KUKA KRL program: p01drop1_s1.src, p01drop1_s1.dat

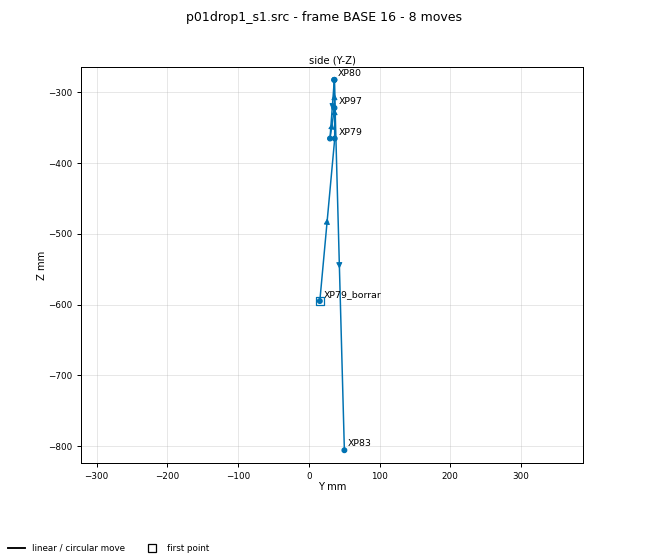
[picture p0: tool path of p01drop1_s1.src in frame BASE 16, 8 of 12 moves have a stored position in this frame; points joined in program order, loops and branches not executed]
--- p01drop1_s1.src ---
&ACCESS RVO1
&REL 4753
&PARAM EDITMASK = *
DEF p01drop1_s1( )

;================================================
; MODELO   : BALANCINA VIEJA
; IE GRUPO : FIP
; ESTACION : ST101
; ROBOT    : 101R1
; FUNCION  : DROP IP
;================================================

;FOLD INI
  ;FOLD BASISTECH INI
    GLOBAL INTERRUPT DECL 3 WHEN $STOPMESS==TRUE DO IR_STOPM ( )
    INTERRUPT ON 3
    BAS (#INITMOV,0 )
  ;ENDFOLD (BASISTECH INI)
;FOLD SPOTTECH INI
;USERSPOT(#INIT)
;ENDFOLD (SPOTTECH INI)
;FOLD GRIPPERTECH INI
USER_GRP(0,DUMMY,DUMMY,GDEFAULT)
INTERRUPT DECL 20 WHEN $FLAG[20]==FALSE DO GRPS(#MON_ERR,20)
;ENDFOLD (GRIPPERTECH INI)
  ;FOLD USER INI
    ;Make your modifications here

  ;ENDFOLD (USER INI)
;ENDFOLD (INI)

;ENTRAR_DEDOS()
;CERRAR_DEDOS()
;ENTRAR_RODILLO()
;ABRIR_CILINDRO_IP()
;CLAMPAR_GONDOLA()
o_type_req=FALSE

;INICIALIZACION GRIPER

;wait area

;FOLD PTP P77 Vel=100 % PDAT22 Tool[13] Base[0];%{PE}%R 5.6.13,%MKUKATPBASIS,%CMOVE,%VPTP,%P 1:PTP, 2:P77, 3:, 5:100, 7:PDAT22
$BWDSTART=FALSE
PDAT_ACT=PPDAT22
FDAT_ACT=FP77
BAS(#PTP_PARAMS,100)
PTP XP77
;ENDFOLD
;FOLD FORDTECH.Area_Req 2 Safety Position, 0 Return To Home, 0 ;%{PE}%MKUKATPUSER
;Area_Req (2,0,0)
wait for $in[18]
$out[18]=false
;ENDFOLD

;TRAYECTORIA DE ENTRADA


;===========================================================
;POSICION FOTO 1 (selccionar esta linea para repetir foto 1)
;===========================================================
;FOLD OUT 38 'PETICION A DISPOSITIVO 6' State=FALSE ;%{PE}%R 5.6.13,%MKUKATPBASIS,%COUT,%VOUTX,%P 2:38, 3:PETICION A DISPOSITIVO 6, 5:FALSE, 6:
$OUT[38]=FALSE
;ENDFOLD
;wait for false


;FOLD PTP P85 Vel=100 % PDAT27 Tool[14]:camara Base[14]:ems_sup;%{PE}%R 5.6.13,%MKUKATPBASIS,%CMOVE,%VPTP,%P 1:PTP, 2:P85, 3:, 5:100, 7:PDAT27
$BWDSTART=FALSE
PDAT_ACT=PPDAT27
FDAT_ACT=FP85
BAS(#PTP_PARAMS,100)
PTP XP85
;ENDFOLD

;FOLD WAIT Time=0.3 sec;%{PE}%R 5.6.13,%MKUKATPBASIS,%CWAIT,%VWAIT,%P 2:0.3
WAIT SEC 0.3
;ENDFOLD

;CHEQUEO SEÑALES RESETEADAS
MAFELEC_TECH (#CHECK_RESET, 8,0,0)

;PIDE FOTO
;FOLD FORDTECH.Tool_Rel 2 ;%{PE}%MKUKATPUSER
TOOL_REL (2)
;ENDFOLD

;PIDE CORRECCIONES
MAFELEC_TECH (#TYPE, 8,0,0)

;EVALUA CORRECCIONES
SWITCH I_TYPE_INFO
CASE 2
o_type_req=FALSE
;FOLD FORDTECH.Tool_Req 2 ;%{PE}%MKUKATPUSER
TOOL_REQ (2)
;ENDFOLD
RECAZOEMS()
goto home
case 3
o_type_req=FALSE
rechazo_bal()
GOTO HOME
ENDSWITCH

;APLICA CORRECIONES A LA BASE
base_data[16]=base_data[14]
MAFELEC_TECH (#GET_CORR, 16,0,0)

tool_data[16]=tool_data[14]
;APLICA CORRECCION ANGULO A TOOL
MAFELEC_TECH (#GET_CORR_TOOL,16 ,0,0)

;REGISTRA CORRECCIONES
MAFELEC_TECH (#REG1, 8,0,0)

;FINALIZA PROCESO CORRECCIONES
o_type_req=false
wait for i_type_info==0
;FOLD FORDTECH.Tool_Req 2 ;%{PE}%MKUKATPUSER
TOOL_REQ (2)
;ENDFOLD

;PUNTO SEGUNA FOTO
xP76=xP85
;FOLD PTP P76 Vel=100 % PDAT21 Tool[16]:camara_corregida Base[16]:EMS_SUP_CORREGIDA;%{PE}%R 5.6.13,%MKUKATPBASIS,%CMOVE,%VPTP,%P 1:PTP, 2:P76, 3:, 5:100, 7:PDAT21
$BWDSTART=FALSE
PDAT_ACT=PPDAT21
FDAT_ACT=FP76
BAS(#PTP_PARAMS,100)
PTP XP76
;ENDFOLD

;FOLD WAIT Time=0.3 sec;%{PE}%R 5.6.13,%MKUKATPBASIS,%CWAIT,%VWAIT,%P 2:0.3
WAIT SEC 0.3
;ENDFOLD

;PETICION SEGUNDA FOTO
;FOLD FORDTECH.Tool_Rel 6 ;%{PE}%MKUKATPUSER
TOOL_REL (6)
;ENDFOLD

;PETICION RESULTADO FOTO
MAFELEC_TECH (#TYPE, 8,0,0)

;EVALUA RESULTADO
SWITCH I_TYPE_INFO
CASE 1 ;FOTO OK
o_type_req=false
wait for i_type_info==0
CASE 2
o_type_req=FALSE
;FOLD FORDTECH.Tool_Req 6 ;%{PE}%MKUKATPUSER
TOOL_REQ (6)
;ENDFOLD
;wait for false
RECAZOEMS()
GOTO HOME
case 3
o_type_req=FALSE
rechazo_bal()
goto home
ENDSWITCH

;FINALIZA PROCESO SEGUNDA FOTO
;FOLD FORDTECH.Tool_Req 6 ;%{PE}%MKUKATPUSER
TOOL_REQ (6)
;ENDFOLD

if not i_dry then

;FOLD CHEQUEO LIMITE SEGUNDO OFFSET
;WAIT FOR EMSupbase_OFFSETz>-200
;WAIT FOR EMSupbase_OFFSETz<200
;WAIT FOR EMSupbase_OFFSETx>-200
;WAIT FOR EMSupbase_OFFSETx<200
;WAIT FOR EMSupbase_OFFSETb>-0.400
;WAIT FOR EMSupbase_OFFSETb<0.400
;ENDFOLD
;APLICAMOS OFFSET
;FOLD OFFSET CORR
;BASE_DATA[8].Z=EMSupbase_CORR.Z+EMSupbase_OFFSETz
;BASE_DATA[8].X=EMSupbase_CORR.X+EMSupbase_OFFSETx
;BASE_DATA[8].B=EMSupbase_CORR.B+EMSupbase_OFFSETb
;ENDFOLD
;goto alejandro
;SACAR_DEDOS()
;wait for false

;ACTIVAR TORQ MONITORING
;FOLD TORQMON SetLimits Axis 1: 50 % Axis 2: 40 % Axis 3: 40 % Axis 4: 50 % Axis 5: 40 % Axis 6: 40 %;%{PE}%R 5.6.13,%MKUKATPBASIS,%CTQ_MON,%VTQ_LIMITS,%P 2:TQ_LIMITS, 4:50, 7:40, 10:40, 13:50, 16:40, 19:40
SET_TQ_VALUES (50,40,40,50,40,40)
;ENDFOLD

;TRAYECTORIA ENTRADA A COGIDA

;FOLD LIN P79_borrar Vel=2 m/s CPDAT21 Tool[16]:camara_corregida Base[16]:EMS_SUP_CORREGIDA;%{PE}%R 5.6.13,%MKUKATPBASIS,%CMOVE,%VLIN,%P 1:LIN, 2:P79_borrar, 3:, 5:2, 7:CPDAT21
$BWDSTART=FALSE
LDAT_ACT=LCPDAT21
FDAT_ACT=FP79_borrar
BAS(#CP_PARAMS,2)
LIN XP79_borrar
;ENDFOLD

;FOLD LIN P79 Vel=2 m/s CPDAT10 Tool[16]:camara_corregida Base[16]:EMS_SUP_CORREGIDA;%{PE}%R 5.6.13,%MKUKATPBASIS,%CMOVE,%VLIN,%P 1:LIN, 2:P79, 3:, 5:2, 7:CPDAT10
$BWDSTART=FALSE
LDAT_ACT=LCPDAT10
FDAT_ACT=FP79
BAS(#CP_PARAMS,2)
LIN XP79
;ENDFOLD

;ABRE CLAMPAS
ABRIR_DEDOS()

;MOVIMIENTO A PUNTO DEJADA
if false then
;FOLD LIN P80 Vel=2 m/s CPDAT11 Tool[16]:camara_corregida Base[16]:EMS_SUP_CORREGIDA;%{PE}%R 5.6.13,%MKUKATPBASIS,%CMOVE,%VLIN,%P 1:LIN, 2:P80, 3:, 5:2, 7:CPDAT11
$BWDSTART=FALSE
LDAT_ACT=LCPDAT11
FDAT_ACT=FP80
BAS(#CP_PARAMS,2)
LIN XP80
;ENDFOLD
endif

;FOLD LIN P98 Vel=2 m/s CPDAT18 Tool[16]:camara_corregida Base[16]:EMS_SUP_CORREGIDA;%{PE}%R 5.6.13,%MKUKATPBASIS,%CMOVE,%VLIN,%P 1:LIN, 2:P98, 3:, 5:2, 7:CPDAT18
$BWDSTART=FALSE
LDAT_ACT=LCPDAT18
FDAT_ACT=FP98
BAS(#CP_PARAMS,2)
LIN XP98
;ENDFOLD
;FOLD LIN P97 Vel=2 m/s CPDAT17 Tool[16]:camara_corregida Base[16]:EMS_SUP_CORREGIDA;%{PE}%R 5.6.13,%MKUKATPBASIS,%CMOVE,%VLIN,%P 1:LIN, 2:P97, 3:, 5:2, 7:CPDAT17
$BWDSTART=FALSE
LDAT_ACT=LCPDAT17
FDAT_ACT=FP97
BAS(#CP_PARAMS,2)
LIN XP97
;ENDFOLD

;FOLD LIN P95 Vel=1 m/s CPDAT15 Tool[16]:camara_corregida Base[16]:EMS_SUP_CORREGIDA;%{PE}%R 5.6.13,%MKUKATPBASIS,%CMOVE,%VLIN,%P 1:LIN, 2:P95, 3:, 5:1, 7:CPDAT15
$BWDSTART=FALSE
LDAT_ACT=LCPDAT15
FDAT_ACT=FP95
BAS(#CP_PARAMS,1)
LIN XP95
;ENDFOLD

;CIERRA CLAMPAS
if not B_EMSdry then
CERRAR_DEDOS()
endif

;FOLD WAIT Time=1 sec;%{PE}%R 5.6.13,%MKUKATPBASIS,%CWAIT,%VWAIT,%P 2:1
WAIT SEC 1
;ENDFOLD

;FOLD LIN P96 Vel=1 m/s CPDAT16 Tool[16]:camara_corregida Base[16]:EMS_SUP_CORREGIDA;%{PE}%R 5.6.13,%MKUKATPBASIS,%CMOVE,%VLIN,%P 1:LIN, 2:P96, 3:, 5:1, 7:CPDAT16
$BWDSTART=FALSE
LDAT_ACT=LCPDAT16
FDAT_ACT=FP96
BAS(#CP_PARAMS,1)
LIN XP96
;ENDFOLD

IF false THEN
;CHEQUEA CLAMPAS CERRADAS
ENDIF
if false then
endif

;ESPERA RESULTADOS CAMARAS ACIMUT Y VOLANTE
;FOLD FORDTECH.Tool_Rel 3 ;%{PE}%MKUKATPUSER
TOOL_REL (3)
;ENDFOLD
;FOLD FORDTECH.Tool_Req 3 ;%{PE}%MKUKATPUSER
TOOL_REQ (3)
;ENDFOLD

if not B_EMSdry then
;ABRE GARRA PARA SOLTAR IP

ABRIR_CILINDRO_IP()
endif

if B_EMSdry then
;punto interdio para liberar orejetas
endif

;FOLD LIN P83 Vel=1 m/s CPDAT13 Tool[16]:camara_corregida Base[16]:EMS_SUP_CORREGIDA;%{PE}%R 5.6.13,%MKUKATPBASIS,%CMOVE,%VLIN,%P 1:LIN, 2:P83, 3:, 5:1, 7:CPDAT13
$BWDSTART=FALSE
LDAT_ACT=LCPDAT13
FDAT_ACT=FP83
BAS(#CP_PARAMS,1)
LIN XP83
;ENDFOLD
;MOVIMIENTO SALIDA
alejandro:

endif

if i_dry then
;FOLD FORDTECH.Tool_Rel 3 ;%{PE}%MKUKATPUSER
TOOL_REL (3)
;ENDFOLD
;FOLD FORDTECH.Tool_Req 3 ;%{PE}%MKUKATPUSER
TOOL_REQ (3)
;ENDFOLD
endif

;DEJA TORQ MONITORING EN VALORES NOMINALES
;FOLD TORQMON SetDefault;%{PE}%R 5.6.13,%MKUKATPBASIS,%CTQ_MON,%VTQ_DEFAULT,%P 2:TQ_DEFAULT
SET_TQ_VALUES ( )
;ENDFOLD

;TRAYECTORIA SALIDA AREA

;wait area ems
;FOLD PTP P89 Vel=100 % PDAT30 Tool[12] Base[0];%{PE}%R 5.6.13,%MKUKATPBASIS,%CMOVE,%VPTP,%P 1:PTP, 2:P89, 3:, 5:100, 7:PDAT30
$BWDSTART=FALSE
PDAT_ACT=PPDAT30
FDAT_ACT=FP89
BAS(#PTP_PARAMS,100)
PTP XP89
;ENDFOLD

;AREA LIBRE Y TRABAJO REALIZADO
;FOLD FORDTECH.Job_Rdy 2 , 1 ;%{PE}%MKUKATPUSER
JOB_READY (2,1)
;ENDFOLD
;FOLD FORDTECH.Area_Rel 2 ;%{PE}%MKUKATPUSER
AREA_REL (2)
;ENDFOLD




home:


END

--- p01drop1_s1.dat ---
&ACCESS RVO1
&REL 4753
&PARAM EDITMASK = *
DEFDAT  P01DROP1_S1
;FOLD EXTERNAL DECLARATIONS;%{PE}%MKUKATPBASIS,%CEXT,%VCOMMON,%P
;FOLD GRIPPERTECH EXT
EXT  H50 (INT  :IN,INT  :IN,INT  :IN,GRP_TYP  :IN )
;ENDFOLD (GRIPPERTECH EXT)
;FOLD SPOTTECH EXT
EXT  USERSPOT (S_COMMAND  :IN,SPOT_TYPE  :IN )
;ENDFOLD (SPOTTECH EXT)
;FOLD BASISTECH EXT;%{PE}%MKUKATPBASIS,%CEXT,%VEXT,%P
EXT  BAS (BAS_COMMAND  :IN,REAL  :IN )
DECL INT SUCCESS
;ENDFOLD (BASISTECH EXT)
;FOLD USER EXT;%{E}%MKUKATPUSER,%CEXT,%VEXT,%P
;Make here your modifications

;ENDFOLD (USER EXT)
;ENDFOLD (EXTERNAL DECLARATIONS)
DECL BASIS_SUGG_T LAST_BASIS={POINT1[] "P100b                   ",POINT2[] "P100b                   ",CP_PARAMS[] "CPDAT21                 ",PTP_PARAMS[] "PDAT36                  ",CONT[] "                        ",CP_VEL[] "2                       ",PTP_VEL[] "100                     ",SYNC_PARAMS[] "SYNCDAT                 ",SPL_NAME[] "S0                      "}
DECL E6POS XP1={X 1562.28699,Y 893.286072,Z 1286.09595,A -15.2613897,B 0.657847583,C -90.4761429,S 2,T 3,E1 0.0,E2 0.0,E3 0.0,E4 0.0,E5 0.0,E6 0.0}
DECL FDAT FP1={TOOL_NO 10,BASE_NO 0,IPO_FRAME #BASE,POINT2[] " ",TQ_STATE FALSE}
DECL PDAT PPDAT1={VEL 100.0,ACC 100.0,APO_DIST 100.0,APO_MODE #CPTP}
DECL E6POS XP2={X 0.052320879,Y -135.084106,Z 32.6104889,A 0.252467006,B -0.648865819,C 1.13480794,S 2,T 3,E1 0.0,E2 0.0,E3 0.0,E4 0.0,E5 0.0,E6 0.0}
DECL FDAT FP2={TOOL_NO 10,BASE_NO 8,IPO_FRAME #BASE,POINT2[] " ",TQ_STATE FALSE}
DECL PDAT PPDAT2={VEL 100.0,ACC 100.0,APO_DIST 100.0}
DECL E6POS XP3={X -0.226943403,Y -135.580994,Z 57.4539795,A 0.252323091,B -0.648702681,C 1.13486397,S 2,T 3,E1 0.0,E2 0.0,E3 0.0,E4 0.0,E5 0.0,E6 0.0}
DECL FDAT FP3={TOOL_NO 10,BASE_NO 8,IPO_FRAME #BASE,POINT2[] " ",TQ_STATE FALSE}
DECL PDAT PPDAT3={VEL 100.0,ACC 100.0,APO_DIST 100.0}
DECL E6POS XP4={X 917.980408,Y 1082.76501,Z 1563.30298,A -10.58006,B -0.816496015,C -90.0786209,S 2,T 3,E1 0.0,E2 0.0,E3 0.0,E4 0.0,E5 0.0,E6 0.0}
DECL FDAT FP4={TOOL_NO 3,BASE_NO 0,IPO_FRAME #BASE,POINT2[] " ",TQ_STATE FALSE}
DECL PDAT PPDAT4={VEL 100.0,ACC 100.0,APO_DIST 100.0,APO_MODE #CPTP}
DECL PDAT PPDAT5={VEL 100.0,ACC 100.0,APO_DIST 100.0}
DECL E6POS XP55={X 669.274719,Y 1258.45898,Z 1571.16199,A 1.68324995,B 0.417000502,C -88.9230118,S 2,T 11,E1 0.0,E2 0.0,E3 0.0,E4 0.0,E5 0.0,E6 0.0}
DECL FDAT FP55={TOOL_NO 3,BASE_NO 0,IPO_FRAME #BASE,POINT2[] " ",TQ_STATE FALSE}
DECL PDAT PPDAT6={VEL 100.0,ACC 100.0,APO_DIST 100.0}
DECL LDAT LCPDAT3={VEL 2.0,ACC 100.0,APO_DIST 100.0,APO_FAC 50.0,ORI_TYP #VAR,CIRC_TYP #BASE,JERK_FAC 50.0,EXAX_IGN 0}
DECL E6POS XP56={X 3.78204703,Y -128.492996,Z -299.213898,A 0.252413303,B -0.64881891,C 1.13486505,S 2,T 3,E1 0.0,E2 0.0,E3 0.0,E4 0.0,E5 0.0,E6 0.0}
DECL FDAT FP56={TOOL_NO 10,BASE_NO 8,IPO_FRAME #BASE,POINT2[] " ",TQ_STATE FALSE}
DECL PDAT PPDAT7={VEL 100.0,ACC 100.0,APO_DIST 50.0,APO_MODE #CPTP}
DECL E6POS XP57={X 825.400024,Y 974.496826,Z 1563.53699,A -6.83336401,B -0.817213476,C -90.0786514,S 2,T 3,E1 0.0,E2 0.0,E3 0.0,E4 0.0,E5 0.0,E6 0.0}
DECL FDAT FP57={TOOL_NO 3,BASE_NO 0,IPO_FRAME #BASE,POINT2[] " ",TQ_STATE FALSE}
DECL PDAT PPDAT8={VEL 100.0,ACC 100.0,APO_DIST 100.0}
DECL LDAT LCPDAT1={VEL 2.0,ACC 100.0,APO_DIST 100.0,APO_FAC 50.0,ORI_TYP #VAR,CIRC_TYP #BASE,JERK_FAC 50.0,EXAX_IGN 0}
DECL E6POS XP58={X 6.92813683,Y -122.939102,Z -579.260681,A 0.251890212,B -0.648669422,C 1.13512194,S 2,T 11,E1 0.0,E2 0.0,E3 0.0,E4 0.0,E5 0.0,E6 0.0}
DECL FDAT FP58={TOOL_NO 3,BASE_NO 8,IPO_FRAME #BASE,POINT2[] " ",TQ_STATE FALSE}
DECL LDAT LCPDAT2={VEL 2.0,ACC 100.0,APO_DIST 100.0,APO_FAC 50.0,ORI_TYP #VAR,CIRC_TYP #BASE,JERK_FAC 50.0,EXAX_IGN 0}
DECL E6POS XP59={X 1195.93005,Y 946.286804,Z 1558.15601,A -25.4987297,B -0.698007703,C -90.0127335,S 2,T 3,E1 0.0,E2 0.0,E3 0.0,E4 0.0,E5 0.0,E6 0.0}
DECL FDAT FP59={TOOL_NO 3,BASE_NO 0,IPO_FRAME #BASE,POINT2[] " ",TQ_STATE FALSE}
DECL PDAT PPDAT9={VEL 100.0,ACC 100.0,APO_DIST 100.0,APO_MODE #CPTP}
DECL E6POS XP60={X 1607.74902,Y 781.598511,Z 1575.47095,A -48.1744194,B -1.694278,C -88.870842,S 2,T 2,E1 0.0,E2 0.0,E3 0.0,E4 0.0,E5 0.0,E6 0.0}
DECL FDAT FP60={TOOL_NO 3,BASE_NO 0,IPO_FRAME #BASE,POINT2[] " ",TQ_STATE FALSE}
DECL PDAT PPDAT10={VEL 100.0,ACC 100.0,APO_DIST 100.0,APO_MODE #CPTP}
DECL E6POS XP61={X 2.21973109,Y 78.0449219,Z -473.749786,A 0.453805208,B -1.02935696,C 1.12841296,S 2,T 11,E1 0.0,E2 0.0,E3 0.0,E4 0.0,E5 0.0,E6 0.0}
DECL FDAT FP61={TOOL_NO 10,BASE_NO 6,IPO_FRAME #BASE,POINT2[] " ",TQ_STATE FALSE}
DECL PDAT PPDAT11={VEL 100.0,ACC 100.0,APO_DIST 100.0}
DECL E6POS XP62={X 686.276306,Y 1072.54199,Z 1338.49402,A -3.73349309,B -0.516365111,C -90.2921371,S 2,T 3,E1 0.0,E2 0.0,E3 0.0,E4 0.0,E5 0.0,E6 0.0}
DECL FDAT FP62={TOOL_NO 10,BASE_NO 0,IPO_FRAME #BASE,POINT2[] " ",TQ_STATE FALSE}
DECL PDAT PPDAT12={VEL 100.0,ACC 100.0,APO_DIST 100.0,APO_MODE #CPTP}
DECL E6POS XP63={X 4.17468405,Y -128.584198,Z -273.346893,A 0.318527609,B -0.649609089,C 1.13304698,S 2,T 11,E1 0.0,E2 0.0,E3 0.0,E4 0.0,E5 0.0,E6 0.0}
DECL FDAT FP63={TOOL_NO 3,BASE_NO 8,IPO_FRAME #BASE,POINT2[] " ",TQ_STATE FALSE}
DECL PDAT PPDAT13={VEL 100.0,ACC 100.0,APO_DIST 100.0,APO_MODE #CPTP}
DECL E6POS XP64={X 141.040298,Y -131.536896,Z -626.476685,A -0.01522478,B 7.10692596,C 0.110732399,S 2,T 3,E1 0.0,E2 0.0,E3 0.0,E4 0.0,E5 0.0,E6 0.0}
DECL FDAT FP64={TOOL_NO 3,BASE_NO 8,IPO_FRAME #BASE,POINT2[] " ",TQ_STATE FALSE}
DECL PDAT PPDAT14={VEL 100.0,ACC 100.0,APO_DIST 100.0,APO_MODE #CPTP}
DECL E6POS XP65={X 1145.12195,Y 865.575378,Z 1562.22705,A -24.1379299,B -0.725280404,C -90.2146072,S 2,T 2,E1 0.0,E2 0.0,E3 0.0,E4 0.0,E5 0.0,E6 0.0}
DECL FDAT FP65={TOOL_NO 3,BASE_NO 0,IPO_FRAME #BASE,POINT2[] " ",TQ_STATE FALSE}
DECL PDAT PPDAT15={VEL 100.0,ACC 100.0,APO_DIST 100.0,APO_MODE #CPTP}
DECL E6POS XP66={X 2.245502,Y 78.0254288,Z -473.714996,A 0.452297091,B -1.028229,C 1.12880397,S 2,T 11,E1 0.0,E2 0.0,E3 0.0,E4 0.0,E5 0.0,E6 0.0}
DECL FDAT FP66={TOOL_NO 10,BASE_NO 8,IPO_FRAME #BASE,POINT2[] " ",TQ_STATE FALSE}
DECL PDAT PPDAT16={VEL 100.0,ACC 100.0,APO_DIST 100.0,APO_MODE #CPTP}
DECL E6POS XP67={X 0.474618286,Y -135.130203,Z 56.3668594,A 0.318735003,B -0.650003672,C 1.133497,S 2,T 3,E1 0.0,E2 0.0,E3 0.0,E4 0.0,E5 0.0,E6 0.0}
DECL FDAT FP67={TOOL_NO 3,BASE_NO 8,IPO_FRAME #BASE,POINT2[] " ",TQ_STATE FALSE}
DECL LDAT LCPDAT4={VEL 2.0,ACC 100.0,APO_DIST 100.0,APO_FAC 50.0,ORI_TYP #VAR,CIRC_TYP #BASE,JERK_FAC 50.0,EXAX_IGN 0}
DECL E6POS XP68={X 2.50332093,Y -131.528702,Z -125.126297,A 0.318527102,B -0.649853289,C 1.13311696,S 2,T 11,E1 0.0,E2 0.0,E3 0.0,E4 0.0,E5 0.0,E6 0.0}
DECL FDAT FP68={TOOL_NO 3,BASE_NO 8,IPO_FRAME #BASE,POINT2[] " ",TQ_STATE FALSE}
DECL LDAT LCPDAT5={VEL 2.0,ACC 100.0,APO_DIST 100.0,APO_FAC 50.0,ORI_TYP #VAR,CIRC_TYP #BASE,JERK_FAC 50.0,EXAX_IGN 0}
DECL E6POS XP69={X 2768.47705,Y 6.94654799,Z 2006.30298,A -150.0289,B 15.6658697,C -84.9255676,S 2,T 43,E1 0.0,E2 0.0,E3 0.0,E4 0.0,E5 0.0,E6 0.0}
DECL FDAT FP69={TOOL_NO 3,BASE_NO 0,IPO_FRAME #BASE,POINT2[] " ",TQ_STATE FALSE}
DECL PDAT PPDAT17={VEL 100.0,ACC 100.0,APO_DIST 100.0,APO_MODE #CPTP}
DECL E6POS XP70={X 2181.64502,Y 940.81012,Z 1193.08899,A -55.6323204,B 0.397260487,C -90.4529495,S 2,T 10,E1 0.0,E2 0.0,E3 0.0,E4 0.0,E5 0.0,E6 0.0}
DECL FDAT FP70={TOOL_NO 10,BASE_NO 0,IPO_FRAME #BASE,POINT2[] " ",TQ_STATE FALSE}
DECL PDAT PPDAT18={VEL 100.0,ACC 100.0,APO_DIST 100.0,APO_MODE #CPTP}
DECL E6POS XP71={X 682.504395,Y 1586.74194,Z 1564.78699,A 0.650965273,B -0.740677118,C -89.7750626,S 2,T 3,E1 0.0,E2 0.0,E3 0.0,E4 0.0,E5 0.0,E6 0.0}
DECL FDAT FP71={TOOL_NO 3,BASE_NO 0,IPO_FRAME #BASE,POINT2[] " ",TQ_STATE FALSE}
DECL LDAT LCPDAT7={VEL 2.0,ACC 100.0,APO_DIST 100.0,APO_FAC 50.0,ORI_TYP #VAR,CIRC_TYP #BASE,JERK_FAC 50.0,EXAX_IGN 0}
DECL LDAT LCPDAT8={VEL 2.0,ACC 100.0,APO_DIST 100.0,APO_FAC 50.0,ORI_TYP #VAR,CIRC_TYP #BASE,JERK_FAC 50.0,EXAX_IGN 0}
DECL E6POS XP72={X 0.052320879,Y -135.084106,Z 32.6104889,A 0.252467006,B -0.648865819,C 1.13480794,S 2,T 3,E1 0.0,E2 0.0,E3 0.0,E4 0.0,E5 0.0,E6 0.0}
DECL FDAT FP72={TOOL_NO 10,BASE_NO 8,IPO_FRAME #BASE,POINT2[] " ",TQ_STATE FALSE}
DECL E6POS XP73={X 0.149559602,Y -134.919601,Z 24.4487591,A 0.252554208,B -0.648425877,C 1.13475394,S 2,T 3,E1 0.0,E2 0.0,E3 0.0,E4 0.0,E5 0.0,E6 0.0}
DECL FDAT FP73={TOOL_NO 10,BASE_NO 8,IPO_FRAME #BASE,POINT2[] " ",TQ_STATE FALSE}
DECL LDAT LCPDAT9={VEL 2.0,ACC 100.0,APO_DIST 100.0,APO_FAC 50.0,ORI_TYP #VAR,CIRC_TYP #BASE,JERK_FAC 50.0,EXAX_IGN 0}
DECL E6POS XP74={X 177.492004,Y 2082.823,Z 1702.56897,A -0.50292927,B 45.5188103,C 179.499405,S 2,T 11,E1 0.0,E2 0.0,E3 0.0,E4 0.0,E5 0.0,E6 0.0}
DECL FDAT FP74={TOOL_NO 0,BASE_NO 0,IPO_FRAME #BASE,POINT2[] " ",TQ_STATE FALSE}
DECL PDAT PPDAT19={VEL 100.0,ACC 100.0,APO_DIST 100.0}
DECL E6POS XP75={X -125.971199,Y -265.283813,Z -316.319305,A 90.6103363,B -1.78813803,C -0.124596797,S 2,T 10,E1 0.0,E2 0.0,E3 0.0,E4 0.0,E5 0.0,E6 0.0}
DECL FDAT FP75={TOOL_NO 8,BASE_NO 14,IPO_FRAME #BASE,POINT2[] " ",TQ_STATE FALSE}
DECL PDAT PPDAT20={VEL 100.0,ACC 100.0,APO_DIST 100.0}
DECL E6POS XP76={X -128.091095,Y 0.680960417,Z -757.682922,A 89.7646408,B -0.642541885,C 0.220073298,S 2,T 11,E1 0.0,E2 0.0,E3 0.0,E4 0.0,E5 0.0,E6 0.0}
DECL FDAT FP76={TOOL_NO 16,BASE_NO 16,IPO_FRAME #BASE,POINT2[] " ",TQ_STATE FALSE}
DECL PDAT PPDAT21={VEL 100.0,ACC 100.0,APO_DIST 100.0}
DECL E6POS XP77={X 705.314392,Y 2000.59497,Z 1624.87805,A -13.2357502,B 44.7311783,C 178.321304,S 2,T 11,E1 0.0,E2 0.0,E3 0.0,E4 0.0,E5 0.0,E6 0.0}
DECL FDAT FP77={TOOL_NO 13,BASE_NO 0,IPO_FRAME #BASE,POINT2[] " ",TQ_STATE FALSE}
DECL PDAT PPDAT22={VEL 100.0,ACC 100.0,APO_DIST 100.0}
DECL E6POS XP78={X 224.640701,Y 2078.11694,Z 1675.72803,A -0.294790298,B 45.0043297,C 179.436996,S 2,T 11,E1 0.0,E2 0.0,E3 0.0,E4 0.0,E5 0.0,E6 0.0}
DECL FDAT FP78={TOOL_NO 0,BASE_NO 0,IPO_FRAME #BASE,POINT2[] " ",TQ_STATE FALSE}
DECL PDAT PPDAT23={VEL 100.0,ACC 100.0,APO_DIST 100.0}
DECL E6POS XP79={X -130.524094,Y 36.7159882,Z -365.105804,A 89.8188171,B -1.25319099,C 0.0377966203,S 2,T 11,E1 0.0,E2 0.0,E3 0.0,E4 0.0,E5 0.0,E6 0.0}
DECL FDAT FP79={TOOL_NO 16,BASE_NO 16,IPO_FRAME #BASE,POINT2[] " ",TQ_STATE FALSE}
DECL LDAT LCPDAT10={VEL 2.0,ACC 20.0,APO_DIST 100.0,APO_FAC 50.0,ORI_TYP #VAR,CIRC_TYP #BASE,JERK_FAC 50.0,EXAX_IGN 0}
DECL E6POS XP80={X -134.476898,Y 36.1417999,Z -282.15741,A 89.8160934,B -1.10210598,C -0.134312794,S 2,T 11,E1 0.0,E2 0.0,E3 0.0,E4 0.0,E5 0.0,E6 0.0}
DECL FDAT FP80={TOOL_NO 16,BASE_NO 16,IPO_FRAME #BASE,POINT2[] " ",TQ_STATE FALSE}
DECL LDAT LCPDAT11={VEL 2.0,ACC 20.0,APO_DIST 100.0,APO_FAC 50.0,ORI_TYP #VAR,CIRC_TYP #BASE,JERK_FAC 50.0,EXAX_IGN 0}
DECL E6POS XP81={X 2576.92993,Y -773.447327,Z -3076.573,A 88.4551315,B -0.226906598,C 91.8414612,S 2,T 10,E1 0.0,E2 0.0,E3 0.0,E4 0.0,E5 0.0,E6 0.0}
DECL FDAT FP81={TOOL_NO 7,BASE_NO 21,IPO_FRAME #BASE,POINT2[] " ",TQ_STATE FALSE}
DECL LDAT LCPDAT12={VEL 2.0,ACC 20.0,APO_DIST 100.0,APO_FAC 50.0,ORI_TYP #VAR,CIRC_TYP #BASE,JERK_FAC 50.0,EXAX_IGN 0}
DECL E6POS XP82={X -112.995796,Y 70.4874191,Z -1061.04797,A 89.9408188,B -1.79147398,C 0.0544125587,S 2,T 10,E1 0.0,E2 0.0,E3 0.0,E4 0.0,E5 0.0,E6 0.0}
DECL FDAT FP82={TOOL_NO 16,BASE_NO 16,IPO_FRAME #BASE,POINT2[] " ",TQ_STATE FALSE}
DECL PDAT PPDAT24={VEL 100.0,ACC 100.0,APO_DIST 100.0}
DECL LDAT LCPDAT13={VEL 2.0,ACC 20.0,APO_DIST 100.0,APO_FAC 50.0,ORI_TYP #VAR,CIRC_TYP #BASE,JERK_FAC 50.0,EXAX_IGN 0}
DECL E6POS XP83={X -130.771606,Y 50.3604202,Z -805.705688,A 89.8190994,B -1.25311804,C 0.0378480516,S 2,T 11,E1 0.0,E2 0.0,E3 0.0,E4 0.0,E5 0.0,E6 0.0}
DECL FDAT FP83={TOOL_NO 16,BASE_NO 16,IPO_FRAME #BASE,POINT2[] " ",TQ_STATE FALSE}
DECL E6POS XP84={X 2360.92407,Y -767.722412,Z -3069.61206,A 88.4529495,B -0.225749105,C 91.8408737,S 2,T 10,E1 0.0,E2 0.0,E3 0.0,E4 0.0,E5 0.0,E6 0.0}
DECL FDAT FP84={TOOL_NO 7,BASE_NO 21,IPO_FRAME #BASE,POINT2[] " ",TQ_STATE FALSE}
DECL LDAT LCPDAT14={VEL 2.0,ACC 20.0,APO_DIST 100.0,APO_FAC 50.0,ORI_TYP #VAR,CIRC_TYP #BASE,JERK_FAC 50.0,EXAX_IGN 0}
DECL E6POS XP85={X -128.091095,Y 0.680960417,Z -757.682922,A 89.7646408,B -0.642541885,C 0.220073298,S 2,T 11,E1 0.0,E2 0.0,E3 0.0,E4 0.0,E5 0.0,E6 0.0}
DECL FDAT FP85={TOOL_NO 14,BASE_NO 14,IPO_FRAME #BASE,POINT2[] " ",TQ_STATE FALSE}
DECL PDAT PPDAT25={VEL 100.0,ACC 100.0,APO_DIST 100.0}
DECL E6POS XP86={X -291.420898,Y 304.775909,Z -863.177612,A 90.2181931,B 1.14026403,C -0.598465204,S 2,T 11,E1 0.0,E2 0.0,E3 0.0,E4 0.0,E5 0.0,E6 0.0}
DECL FDAT FP86={TOOL_NO 14,BASE_NO 14,IPO_FRAME #BASE,POINT2[] " ",TQ_STATE FALSE}
DECL PDAT PPDAT26={VEL 100.0,ACC 100.0,APO_DIST 100.0}
DECL LDAT LCPDAT15={VEL 2.0,ACC 100.0,APO_DIST 100.0,APO_FAC 50.0,ORI_TYP #VAR,CIRC_TYP #BASE,JERK_FAC 50.0,EXAX_IGN 0}
DECL PDAT PPDAT27={VEL 100.0,ACC 100.0,APO_DIST 100.0}
DECL E6POS XP87={X 637.203308,Y 1990.72998,Z 1675.72803,A -11.87428,B 45.0043297,C 179.436996,S 2,T 11,E1 0.0,E2 0.0,E3 0.0,E4 0.0,E5 0.0,E6 0.0}
DECL FDAT FP87={TOOL_NO 0,BASE_NO 0,IPO_FRAME #BASE,POINT2[] " ",TQ_STATE FALSE}
DECL PDAT PPDAT28={VEL 100.0,ACC 100.0,APO_DIST 100.0}
DECL E6POS XP88={X -128.091095,Y 0.680960417,Z -757.682922,A 89.7646408,B -0.642541885,C 0.220073298,S 2,T 11,E1 0.0,E2 0.0,E3 0.0,E4 0.0,E5 0.0,E6 0.0}
DECL FDAT FP88={TOOL_NO 14,BASE_NO 14,IPO_FRAME #BASE,POINT2[] " ",TQ_STATE FALSE}
DECL PDAT PPDAT29={VEL 100.0,ACC 100.0,APO_DIST 100.0}
DECL PDAT PPDAT30={VEL 100.0,ACC 100.0,APO_DIST 100.0}
DECL E6POS XP89={X 704.915588,Y 2000.79797,Z 1624.86499,A -13.2152596,B 44.7332916,C 178.322906,S 2,T 11,E1 0.0,E2 0.0,E3 0.0,E4 0.0,E5 0.0,E6 0.0}
DECL FDAT FP89={TOOL_NO 12,BASE_NO 0,IPO_FRAME #BASE,POINT2[] " ",TQ_STATE FALSE}
DECL PDAT PPDAT31={VEL 100.0,ACC 100.0,APO_DIST 100.0}
DECL E6POS XP90={X 801.582214,Y 1166.55701,Z 2133.69409,A -36.2449303,B 64.0939331,C -137.098602,S 2,T 11,E1 0.0,E2 0.0,E3 0.0,E4 0.0,E5 0.0,E6 0.0}
DECL FDAT FP90={TOOL_NO 0,BASE_NO 0,IPO_FRAME #BASE,POINT2[] " ",TQ_STATE FALSE}
DECL PDAT PPDAT32={VEL 100.0,ACC 100.0,APO_DIST 100.0}
DECL E6POS XP91={X 981.520325,Y 735.968872,Z 2395.88599,A -60.3835602,B 46.7861595,C -152.051498,S 2,T 11,E1 0.0,E2 0.0,E3 0.0,E4 0.0,E5 0.0,E6 0.0}
DECL FDAT FP91={TOOL_NO 0,BASE_NO 0,IPO_FRAME #BASE,POINT2[] " ",TQ_STATE FALSE}
DECL PDAT PPDAT33={VEL 100.0,ACC 100.0,APO_DIST 100.0}
DECL E6POS XP92={X 946.800476,Y 97.3742676,Z 2526.12598,A -112.670303,B 16.4910603,C -176.548294,S 2,T 11,E1 0.0,E2 0.0,E3 0.0,E4 0.0,E5 0.0,E6 0.0}
DECL FDAT FP92={TOOL_NO 0,BASE_NO 0,IPO_FRAME #BASE,POINT2[] " ",TQ_STATE FALSE}
DECL PDAT PPDAT34={VEL 100.0,ACC 100.0,APO_DIST 100.0}
DECL E6POS XP93={X 946.800476,Y 97.3742676,Z 2526.12598,A -112.670303,B 16.4910603,C -176.548294,S 2,T 11,E1 0.0,E2 0.0,E3 0.0,E4 0.0,E5 0.0,E6 0.0}
DECL FDAT FP93={TOOL_NO 0,BASE_NO 0,IPO_FRAME #BASE,POINT2[] " ",TQ_STATE FALSE}
DECL PDAT PPDAT35={VEL 100.0,ACC 100.0,APO_DIST 100.0}
DECL E6POS XP94={X 946.800476,Y 97.3742676,Z 2526.12598,A -112.670303,B 16.4910603,C -176.548294,S 2,T 11,E1 0.0,E2 0.0,E3 0.0,E4 0.0,E5 0.0,E6 0.0}
DECL FDAT FP94={TOOL_NO 0,BASE_NO 0,IPO_FRAME #BASE,POINT2[] " ",TQ_STATE FALSE}
DECL E6POS XP95={X -134.468307,Y 36.1525993,Z -282.158997,A 89.8184128,B -1.90639997,C -0.134154499,S 2,T 11,E1 0.0,E2 0.0,E3 0.0,E4 0.0,E5 0.0,E6 0.0}
DECL FDAT FP95={TOOL_NO 16,BASE_NO 16,IPO_FRAME #BASE,POINT2[] " ",TQ_STATE FALSE}
DECL E6POS XP96={X -134.476898,Y 36.1417999,Z -282.15741,A 89.8160934,B -1.10210598,C -0.134312794,S 2,T 11,E1 0.0,E2 0.0,E3 0.0,E4 0.0,E5 0.0,E6 0.0}
DECL FDAT FP96={TOOL_NO 16,BASE_NO 16,IPO_FRAME #BASE,POINT2[] " ",TQ_STATE FALSE}
DECL LDAT LCPDAT16={VEL 2.0,ACC 100.0,APO_DIST 100.0,APO_FAC 50.0,ORI_TYP #VAR,CIRC_TYP #BASE,JERK_FAC 50.0,EXAX_IGN 0}
DECL E6POS XP97={X -131.834793,Y 36.3743401,Z -321.795898,A 89.8007507,B -1.174541,C -0.0511082411,S 2,T 11,E1 0.0,E2 0.0,E3 0.0,E4 0.0,E5 0.0,E6 0.0}
DECL FDAT FP97={TOOL_NO 16,BASE_NO 16,IPO_FRAME #BASE,POINT2[] " ",TQ_STATE FALSE}
DECL LDAT LCPDAT17={VEL 2.0,ACC 100.0,APO_DIST 100.0,APO_FAC 50.0,ORI_TYP #VAR,CIRC_TYP #BASE,JERK_FAC 50.0,EXAX_IGN 0}
DECL E6POS XP98={X -130.587799,Y 30.0074806,Z -365.104004,A 89.8171768,B -1.25286901,C 0.0368510187,S 2,T 11,E1 0.0,E2 0.0,E3 0.0,E4 0.0,E5 0.0,E6 0.0}
DECL FDAT FP98={TOOL_NO 16,BASE_NO 16,IPO_FRAME #BASE,POINT2[] " ",TQ_STATE FALSE}
DECL LDAT LCPDAT18={VEL 2.0,ACC 100.0,APO_DIST 100.0,APO_FAC 50.0,ORI_TYP #VAR,CIRC_TYP #BASE,JERK_FAC 50.0,EXAX_IGN 0}
DECL E6POS XP99={X -128.091507,Y 0.682539582,Z -757.687622,A 89.7645035,B -0.642573476,C 0.220033705,S 2,T 11,E1 0.0,E2 0.0,E3 0.0,E4 0.0,E5 0.0,E6 0.0}
DECL FDAT FP99={TOOL_NO 16,BASE_NO 16,IPO_FRAME #BASE,POINT2[] " ",TQ_STATE FALSE}
DECL LDAT LCPDAT19={VEL 2.0,ACC 20.0,APO_DIST 100.0,APO_FAC 50.0,ORI_TYP #VAR,CIRC_TYP #BASE,JERK_FAC 50.0,EXAX_IGN 0}
DECL E6POS XP99B={X -131.541702,Y 29.5267906,Z -332.084412,A 89.8041229,B -1.19263005,C -0.0311941002,S 2,T 11,E1 0.0,E2 0.0,E3 0.0,E4 0.0,E5 0.0,E6 0.0}
DECL FDAT FP99b={TOOL_NO 16,BASE_NO 16,IPO_FRAME #BASE,POINT2[] " ",TQ_STATE FALSE}
DECL PDAT PPDAT36={VEL 100.0,ACC 100.0,APO_DIST 100.0,APO_MODE #CPTP}
DECL LDAT LCPDAT20={VEL 2.0,ACC 20.0,APO_DIST 100.0,APO_FAC 50.0,ORI_TYP #VAR,CIRC_TYP #BASE,JERK_FAC 50.0,EXAX_IGN 0}
DECL LDAT LCPDAT21={VEL 2.0,ACC 20.0,APO_DIST 100.0,APO_FAC 50.0,ORI_TYP #VAR,CIRC_TYP #BASE,JERK_FAC 50.0,EXAX_IGN 0}
DECL E6POS XP100b={X -130.524094,Y 36.7159882,Z -365.105804,A 89.8188171,B -1.25319099,C 0.0377966203,S 2,T 11,E1 0.0,E2 0.0,E3 0.0,E4 0.0,E5 0.0,E6 0.0}
DECL FDAT FP100b={TOOL_NO 16,BASE_NO 16,IPO_FRAME #BASE,POINT2[] " ",TQ_STATE FALSE}
DECL E6POS XP79aborrar={X -129.0914,Y 15.6365004,Z -594.820679,A 89.784462,B -0.897801876,C 0.140368894,S 2,T 11,E1 0.0,E2 0.0,E3 0.0,E4 0.0,E5 0.0,E6 0.0}
DECL FDAT FP79aborrar={TOOL_NO 16,BASE_NO 16,IPO_FRAME #BASE,POINT2[] " ",TQ_STATE FALSE}
DECL E6POS XP79_borrar={X -129.0914,Y 15.6365004,Z -594.820679,A 89.784462,B -0.897801876,C 0.140368894,S 2,T 11,E1 0.0,E2 0.0,E3 0.0,E4 0.0,E5 0.0,E6 0.0}
DECL FDAT FP79_borrar={TOOL_NO 16,BASE_NO 16,IPO_FRAME #BASE,POINT2[] " ",TQ_STATE FALSE}
ENDDAT
